Fanuc KAREL source: kc00053.KL

-- PROVISIONAL review KL for V1013-1; original PC SHA256 eeaaf8e70586c254be00dab927b6867ffbd5ec2ae8abd0874388f7bb3f27c7f7
-- Incomplete behavior may be omitted. Consult companion uncertainty JSON. Do not deploy.
PROGRAM KC00053
%NOLOCKGROUP
BEGIN
  -- UNRESOLVED_PC offsets 5-39; opcodes 27,22,22,22,22,22,31
  -- UNRESOLVED_PC offsets 44-48; opcodes 7F
END KC00053
